// TwinCAT 3 PLC project SynergyPLC
// ProgramVersion: 3.1.4024.12
// libraries:
//   Tc2_EtherCAT, * (Beckhoff Automation GmbH)
//   Tc2_Standard, * (Beckhoff Automation GmbH)
//   Tc2_System, * (Beckhoff Automation GmbH)
//   Tc3_EventLogger, * (Beckhoff Automation GmbH)
//   Tc3_Module, * (Beckhoff Automation GmbH)
//   Tc3_PlasticInterfaceMotion, * (Beckhoff Automation GmbH)
//   Tc3_PlasticInterfaceNc, * (Beckhoff Automation GmbH)
// project tree:
//   GlobalBase/ WatchdogTimer.TcPOU
//   MotionControlBaseAnkur/ AxisBase.TcPOU (excluded from build), ModuleBase.TcPOU (not stored)
//   MotionControlBaseAnkur/DUTs/ Application.TcDUT, AxisData.TcDUT (excluded from build), AxisProperties.TcDUT, AxisStatus.TcDUT (not stored) (excluded from build), GearingType.TcDUT (not stored), Hardware.TcDUT (not stored), HomeFlagType.TcDUT, Homing.TcDUT, HomingMode.TcDUT (not stored), ID.TcDUT, ManualSettings.TcDUT, Mechanical.TcDUT (not stored), OperationLimits.TcDUT (excluded from build), OperationMode.TcDUT (excluded from build), StageBase.TcDUT, StepBase.TcDUT
//   MotionControlBaseAnkur/GVLs/ mcGlobal.TcGVL
//   MotionControlBase/DUTs/ ST_mcAxisNC.TcDUT, E_mcOperationMode.TcTLEO, ST_mcAxisStatus.TcDUT, ST_mcJogAllowance.TcDUT, ST_mcJogParameters.TcDUT, ST_mcAxisOperationLimits.TcDUT
//   MotionControlBase/ FB_mcModulesConfigurator.TcPOU, FB_mcAxisBase.TcPOU, FB_mcAxesConfigurator.TcPOU, FB_mcModuleBase.TcPOU, FB_mcOperationMode.TcPOU
//   MotionControlBase/GVLs/ mcGVL.TcGVL
//   Synergy/GVLs/ synGlobal.TcGVL
//   Synergy/MAIN/ Main1ms.TcPOU
//   / Task1ms.TcTTO
// real-time tasks:
//   TASK Task1ms: cycle T#1ms, priority 1, ADS port 351
// motion (NC):
//   TASK NC-Task 1 SAF: cycle T#1ms, priority 4, ADS port 501
//   TASK NC-Task 1 SVB: cycle T#1ms, priority 8, ADS port 511
//   AXIS Axis 1 (id 1)
//     OtherSettings: AllowMotionCmdToSlave=true
//     encoder EncType=1
//     drive DrvType=5
//       Analog: TorqueSetpointScale=10, ScaleFactorActTorque=0.1
//       TimeComp: TaskDelayCycles=1
//     controller CtrType=1
//       CtrPara: PriorControlFactor=1
//         Observer: BandWidth=20
//   AXIS Axis 2 (id 2)
//     OtherSettings: AllowMotionCmdToSlave=true
//     encoder EncType=1
//     drive DrvType=5
//       Analog: TorqueSetpointScale=10, ScaleFactorActTorque=0.1
//       TimeComp: TaskDelayCycles=1
//     controller CtrType=1
//       CtrPara: PriorControlFactor=1
//         Observer: BandWidth=20
//   AXIS Axis 3 (id 3)
//     OtherSettings: AllowMotionCmdToSlave=true
//     encoder EncType=1
//     drive DrvType=5
//       Analog: TorqueSetpointScale=10, ScaleFactorActTorque=0.1
//       TimeComp: TaskDelayCycles=1
//     controller CtrType=1
//       CtrPara: PriorControlFactor=1
//         Observer: BandWidth=20
//   AXIS Axis 4 (id 4)
//     OtherSettings: AllowMotionCmdToSlave=true
//     encoder EncType=1
//     drive DrvType=5
//       Analog: TorqueSetpointScale=10, ScaleFactorActTorque=0.1
//       TimeComp: TaskDelayCycles=1
//     controller CtrType=1
//       CtrPara: PriorControlFactor=1
//         Observer: BandWidth=20
//   AXIS Axis 5 (id 5)
//     OtherSettings: AllowMotionCmdToSlave=true
//     encoder EncType=1
//     drive DrvType=5
//       Analog: TorqueSetpointScale=10, ScaleFactorActTorque=0.1
//       TimeComp: TaskDelayCycles=1
//     controller CtrType=1
//       CtrPara: PriorControlFactor=1
//         Observer: BandWidth=20
//   AXIS Axis 6 (id 6)
//     OtherSettings: AllowMotionCmdToSlave=true
//     encoder EncType=1
//     drive DrvType=5
//       Analog: TorqueSetpointScale=10, ScaleFactorActTorque=0.1
//       TimeComp: TaskDelayCycles=1
//     controller CtrType=1
//       CtrPara: PriorControlFactor=1
//         Observer: BandWidth=20
//   AXIS Axis 7 (id 7)
//     OtherSettings: AllowMotionCmdToSlave=true
//     encoder EncType=1
//     drive DrvType=5
//       Analog: TorqueSetpointScale=10, ScaleFactorActTorque=0.1
//       TimeComp: TaskDelayCycles=1
//     controller CtrType=1
//       CtrPara: PriorControlFactor=1
//         Observer: BandWidth=20
//   AXIS Axis 8 (id 8)
//     OtherSettings: AllowMotionCmdToSlave=true
//     encoder EncType=1
//     drive DrvType=5
//       Analog: TorqueSetpointScale=10, ScaleFactorActTorque=0.1
//       TimeComp: TaskDelayCycles=1
//     controller CtrType=1
//       CtrPara: PriorControlFactor=1
//         Observer: BandWidth=20
// variable links:
//   SynergyPLC/SynergyPLC Instance <-> NC-Task 1 SAF/Axes/Axis 1
//     Task1ms Inputs/Main1ms.mcModules[1].Axis[1].fbLocalNc.AxisRef.NcToPlc <-> Outputs/ToPlc
//     Task1ms Outputs/Main1ms.mcModules[1].Axis[1].fbLocalNc.AxisRef.PlcToNc <-> Inputs/FromPlc
//   SynergyPLC/SynergyPLC Instance <-> NC-Task 1 SAF/Axes/Axis 2
//     Task1ms Inputs/Main1ms.mcModules[1].Axis[2].fbLocalNc.AxisRef.NcToPlc <-> Outputs/ToPlc
//     Task1ms Outputs/Main1ms.mcModules[1].Axis[2].fbLocalNc.AxisRef.PlcToNc <-> Inputs/FromPlc
//   SynergyPLC/SynergyPLC Instance <-> NC-Task 1 SAF/Axes/Axis 3
//     Task1ms Inputs/Main1ms.mcModules[1].Axis[3].fbLocalNc.AxisRef.NcToPlc <-> Outputs/ToPlc
//     Task1ms Outputs/Main1ms.mcModules[1].Axis[3].fbLocalNc.AxisRef.PlcToNc <-> Inputs/FromPlc
//   SynergyPLC/SynergyPLC Instance <-> NC-Task 1 SAF/Axes/Axis 4
//     Task1ms Inputs/Main1ms.mcModules[1].Axis[4].fbLocalNc.AxisRef.NcToPlc <-> Outputs/ToPlc
//     Task1ms Outputs/Main1ms.mcModules[1].Axis[4].fbLocalNc.AxisRef.PlcToNc <-> Inputs/FromPlc
//   SynergyPLC/SynergyPLC Instance <-> NC-Task 1 SAF/Axes/Axis 5
//     Task1ms Inputs/Main1ms.mcModules[1].Axis[5].fbLocalNc.AxisRef.NcToPlc <-> Outputs/ToPlc
//     Task1ms Outputs/Main1ms.mcModules[1].Axis[5].fbLocalNc.AxisRef.PlcToNc <-> Inputs/FromPlc
//   SynergyPLC/SynergyPLC Instance <-> NC-Task 1 SAF/Axes/Axis 6
//     Task1ms Inputs/Main1ms.mcModules[1].Axis[6].fbLocalNc.AxisRef.NcToPlc <-> Outputs/ToPlc
//     Task1ms Outputs/Main1ms.mcModules[1].Axis[6].fbLocalNc.AxisRef.PlcToNc <-> Inputs/FromPlc
//   SynergyPLC/SynergyPLC Instance <-> NC-Task 1 SAF/Axes/Axis 7
//     Task1ms Inputs/Main1ms.mcModules[1].Axis[7].fbLocalNc.AxisRef.NcToPlc <-> Outputs/ToPlc
//     Task1ms Outputs/Main1ms.mcModules[1].Axis[7].fbLocalNc.AxisRef.PlcToNc <-> Inputs/FromPlc
//   SynergyPLC/SynergyPLC Instance <-> NC-Task 1 SAF/Axes/Axis 8
//     Task1ms Inputs/Main1ms.mcModules[1].Axis[8].fbLocalNc.AxisRef.NcToPlc <-> Outputs/ToPlc
//     Task1ms Outputs/Main1ms.mcModules[1].Axis[8].fbLocalNc.AxisRef.PlcToNc <-> Inputs/FromPlc

CONFIGURATION SynergyPLC
    RESOURCE PLC ON TwinCAT3
        TASK Task1ms(INTERVAL := T#1ms, PRIORITY := 1);
        PROGRAM Main1ms WITH Task1ms : Main1ms;
    END_RESOURCE
END_CONFIGURATION

// ---- MotionControlBaseAnkur/DUTs/Application.TcDUT
TYPE Application :
STRUCT
	GearingType			:	GearingType;
END_STRUCT
END_TYPE

// ---- MotionControlBaseAnkur/DUTs/AxisData.TcDUT
TYPE AxisData :
STRUCT
	lrActPosition			:		LREAL;
	lrActVelocity			:		LREAL;
	lrActTorque				:		LREAL;
	lrMotorTemp				:		LREAL;
END_STRUCT
END_TYPE

// ---- MotionControlBaseAnkur/DUTs/AxisProperties.TcDUT
TYPE AxisProperties :
STRUCT
	stIdentification			:		ID;
	stHardware					:		Hardware;
	stApplication				:		Application;
	stHoming					:		Homing;
	stOperationLimits			:		OperationLimits;
END_STRUCT
END_TYPE

// ---- MotionControlBaseAnkur/DUTs/HomeFlagType.TcDUT
{attribute 'qualified_only'}
{attribute 'strict'}
TYPE HomeFlagType :
(
	eSensor := 1,
	eHardStop := 2
);
END_TYPE

// ---- MotionControlBaseAnkur/DUTs/Homing.TcDUT
TYPE Homing :
STRUCT
	Mode			:		HomingMode;
	FlagType		:		HomeFlagType;
	bHomeInput		:		BOOL;
	rOffset			:		REAL;
	rVelocity		:		REAL;
	rTorque			:		REAL;
END_STRUCT
END_TYPE

// ---- MotionControlBaseAnkur/DUTs/ID.TcDUT
TYPE ID :
STRUCT
	intIndex			:	INT;
	sName				:	STRING;
	intMasterIndex		:	INT;
END_STRUCT
END_TYPE

// ---- MotionControlBaseAnkur/DUTs/ManualSettings.TcDUT
TYPE ManualSettings :
STRUCT
	lrJogVelocity			:		LREAL;
	lrJogRamp				:		LREAL;
	lrJogJerk				:		LREAL;
	lrJogTorque				:		LREAL;
END_STRUCT
END_TYPE

// ---- MotionControlBaseAnkur/DUTs/OperationLimits.TcDUT
TYPE OperationLimits :
STRUCT
	rMinPosition		:		REAL;
	rMaxPosition		:		REAL;
	rMaxVelocity		:		REAL;
	rJogVelocity		:		REAL;
	tMaxMotionTime		:		TIME;
END_STRUCT
END_TYPE

// ---- MotionControlBaseAnkur/DUTs/OperationMode.TcDUT
{attribute 'qualified_only'}
{attribute 'strict'}
TYPE OperationMode :
(
	eManual 	:= 1,
	eService 	:= 2,
	eAutomatic 	:= 3,
	eSimulation := 4
);
END_TYPE

// ---- MotionControlBaseAnkur/DUTs/StageBase.TcDUT
TYPE StageBase :
STRUCT
	bEnable			:		BOOL;
	bTrigger		:		BOOL;
	bMoveActive		:		BOOL;
	tMoveTime		:		TIME;
	intSteps		:		INT;
	Step			:		ARRAY[1..5] OF StepBase;
END_STRUCT
END_TYPE

// ---- MotionControlBaseAnkur/DUTs/StepBase.TcDUT
TYPE StepBase :
STRUCT
	rSetVelocity		:		REAL;
	rSetRamp			:		REAL;
	rSetEndPosition		:		REAL;
END_STRUCT
END_TYPE

// ---- MotionControlBase/DUTs/ST_mcAxisNC.TcDUT
TYPE ST_mcAxisNC :
STRUCT
	lrActPosition			:		LREAL;
	lrActVelocity			:		LREAL;
	lrActTorque				:		LREAL;
	lrMotorTemp				:		LREAL;
END_STRUCT
END_TYPE

// ---- MotionControlBase/DUTs/E_mcOperationMode.TcTLEO
{attribute 'qualified_only'}
{attribute 'strict'}
TYPE E_mcOperationMode : // Operation modes defined
(
	Initialization :=1,
	Service :=2,
	Manual :=3,
	Simulation :=4,
	Automatic :=5
);
END_TYPE

// ---- MotionControlBase/DUTs/ST_mcAxisStatus.TcDUT
TYPE ST_mcAxisStatus :
STRUCT
	bPowerEnabled		:		BOOL; // Power is enabled
	bHomed				:		BOOL; // Homed
	bStandStill			:		BOOL; // Standstill
	bMoving				: 		BOOL; // Moving
	bError				:       BOOL; // Error
END_STRUCT
END_TYPE

// ---- MotionControlBase/DUTs/ST_mcJogAllowance.TcDUT
TYPE ST_mcJogAllowance :
STRUCT
	bAllowJogParameters : BOOL; // Boolean to check if jogging is allowed because of parameters
	bAllowJogOperationMode : BOOL; // Boolean to check if jogging is allowed because of operation mode
END_STRUCT
END_TYPE

// ---- MotionControlBase/DUTs/ST_mcJogParameters.TcDUT
TYPE ST_mcJogParameters :
STRUCT
	lrJogAcceleration		:			LREAL;	//Jog acceleration
	lrJogDeceleration		: 			LREAL;	//Jog deceleration
	lrJogJerkValue			:			LREAL;	//Jog jerk
	lrJogVelocity			:			LREAL;	//Jog velocity
	lrJogLimitPositive		:      		LREAL;  // Jog Positive Torque Limit
	lrJogLimitNegative		:			LREAL;  // Jog Negative Torque Limit
END_STRUCT
END_TYPE

// ---- MotionControlBase/DUTs/ST_mcAxisOperationLimits.TcDUT
TYPE ST_mcAxisOperationLimits :
STRUCT
	lrSoftMinPosition	:			LREAL;	//Minimum position of travel allowed
	lrSoftMaxPosition	: 			LREAL;	//Maximum position of travel allowed
	lrDefaultAcceleration	:		LREAL;	//Maximum Acceleration allowed
	lrDefaultDeceleration	:		LREAL;	//Minimum deceleration allowed
	lrMaxVelocity		:      		LREAL;  //Maximum Velocity allowed
END_STRUCT
END_TYPE

// ---- MotionControlBaseAnkur/GVLs/mcGlobal.TcGVL
{attribute 'qualified_only'}
VAR_GLOBAL
//	fbMotionModule	:		ARRAY[1..cMaxNoOfModule] OF ModuleBase;
END_VAR

VAR_GLOBAL CONSTANT
	cMaxNoOfAxis			:		INT := 8;
	cMinNoOfAxis			:		INT := 1;
	
	cMaxNoOfModule			:		INT := 4;
	cMinNoOfModule			:		INT := 1;
	
	
END_VAR

// ---- MotionControlBase/GVLs/mcGVL.TcGVL
{attribute 'qualified_only'}
VAR_GLOBAL
	OperationMode : FB_MCOperationMode; // Operation mode 
	AxesConfigurator : FB_mcAxesConfigurator; // Configurator to set number of axes
	ModulesConfigurator : FB_mcModulesConfigurator; // Configurator to set number of modules
END_VAR

VAR_GLOBAL CONSTANT
	cMaxAxesCapacity: UINT := 8; // Maximum designed axes capacity by hardware
	cMinAxesCapacity: UINT := 1; // Minimum designed axes capacity by hardware
	cMaxModuleCapacity	: UINT := 4; // Maximum designed modules capacity by hardware
	cMinModuleCapacity	: UINT := 1; // Minimum designed modules capacity by hardware
END_VAR

// ---- Synergy/GVLs/synGlobal.TcGVL
{attribute 'qualified_only'}
VAR_GLOBAL
END_VAR

// ---- Synergy/MAIN/Main1ms.TcPOU
PROGRAM Main1ms
VAR
	mcModules		: ARRAY [1..mcGvl.cMaxModuleCapacity] OF FB_mcModuleBase;
	mcCount			: UINT;
END_VAR

A_mcCyclic();

ACTION A_mcCyclic:
mcGvl.OperationMode(); // Operation mode 
mcGvl.AxesConfigurator(); // Configurator to set number of axes
mcGvl.ModulesConfigurator(); // Configurator to set number of modules

FOR mcCount := 1 TO mcGvl.ModulesConfigurator.uiNoModulesActive DO
	mcModules[mcCount]();
END_FOR;
END_ACTION

END_PROGRAM

// ---- MotionControlBase/FB_mcModuleBase.TcPOU
FUNCTION_BLOCK FB_mcModuleBase
VAR
	Axis			:		ARRAY[1..mcGvl.cMaxAxesCapacity] OF FB_mcAxisBase[
															(AxisName		:=	'Axis1',
															nPtpPoints		:=	5,
															iProcessHandler	:=	0,
															iTorqueLimiting	:=	0,
															iPosCamLookup	:=	0,
															iVeloCamLookup	:=	0,
															iPtpCamLookup	:=	0),
															(AxisName		:=	'Axis2',
															nPtpPoints		:=	5,
															iProcessHandler	:=	0,
															iTorqueLimiting	:=	0,
															iPosCamLookup	:=	0,
															iVeloCamLookup	:=	0,
															iPtpCamLookup	:=	0),
															(AxisName		:=	'Axis3',
															nPtpPoints		:=	5,
															iProcessHandler	:=	0,
															iTorqueLimiting	:=	0,
															iPosCamLookup	:=	0,
															iVeloCamLookup	:=	0,
															iPtpCamLookup	:=	0),
															(AxisName		:=	'Axis4',
															nPtpPoints		:=	5,
															iProcessHandler	:=	0,
															iTorqueLimiting	:=	0,
															iPosCamLookup	:=	0,
															iVeloCamLookup	:=	0,
															iPtpCamLookup	:=	0),
															(AxisName		:=	'Axis5',
															nPtpPoints		:=	5,
															iProcessHandler	:=	0,
															iTorqueLimiting	:=	0,
															iPosCamLookup	:=	0,
															iVeloCamLookup	:=	0,
															iPtpCamLookup	:=	0),
															(AxisName		:=	'Axis6',
															nPtpPoints		:=	5,
															iProcessHandler	:=	0,
															iTorqueLimiting	:=	0,
															iPosCamLookup	:=	0,
															iVeloCamLookup	:=	0,
															iPtpCamLookup	:=	0),
															(AxisName		:=	'Axis7',
															nPtpPoints		:=	5,
															iProcessHandler	:=	0,
															iTorqueLimiting	:=	0,
															iPosCamLookup	:=	0,
															iVeloCamLookup	:=	0,
															iPtpCamLookup	:=	0),
															(AxisName		:=	'Axis8',
															nPtpPoints		:=	5,
															iProcessHandler	:=	0,
															iTorqueLimiting	:=	0,
															iPosCamLookup	:=	0,
															iVeloCamLookup	:=	0,
															iPtpCamLookup	:=	0)
															];
	uiCount				:		UINT;
END_VAR

VAR_INPUT
END_VAR

FOR uiCount := 1 TO mcGVL.AxesConfigurator.uiNoAxesActive DO
	Axis[uiCount].A_Cyclic();
END_FOR

END_FUNCTION_BLOCK

// ---- MotionControlBase/FB_mcAxisBase.TcPOU
FUNCTION_BLOCK FB_mcAxisBase EXTENDS FB_AxisNcBase
VAR_INPUT
	bPowerEnable : BOOL; // Enable Power
	bJogPositive : BOOL; // Jog Positive
	bJogNegative : BOOL; // Jog Negative
	bStop: BOOL; // Stop axis
	bReset: BOOL; // Reset axis
	bExecuteOpLimits: BOOL; // Write operation limits
END_VAR
VAR_OUTPUT
	bBaseFBError : BOOL; // Internal library error
	stStatus: ST_mcAxisStatus; // Status booleans of Axis
	stDataNC: ST_mcAxisNC; // Real data from drive
END_VAR
VAR
	stJogAllowance : ST_mcJogAllowance; // Status bits troubleshooting
	rTrigOpLimits : R_TRIG; // Operation limits trigger
END_VAR

VAR_INPUT PERSISTENT
	stJogParameters : ST_mcJogParameters; // Accel, Decel, Velocity etc
	stOperationLimits : ST_mcAxisOperationLimits; // Soft pos limits, vel limits
END_VAR

VAR CONSTANT 
	cJogMinParameter : REAL := 0.0;  // Minimum parameters for jog to be set to 0 
END_VAR

A_Cyclic(); // Cyclic calls of routines

ACTION A_Cyclic:
SUPER^.Cyclic();						//Cyclic method to initialize underlying motion blocks

IF M_FbError() THEN
;  // Error Exists in Base FB
ELSE  

	// Calling of method to turn power on/off
	M_Power(bCommand:= bPowerEnable);  		
	
	//Calling of method to jog + or - 
	M_Jog(bCommandJogP:= bJogPositive,bCommandJogM:= bJogNegative);

END_IF;

// Calling of method to stop axis
M_Stop(bCommand:= bStop); 

// Calling of method to reset axis
M_Reset(bCommand:= bReset); 

// Calling of method to write operation limits of an axis
rTrigOpLimits(CLK:= bExecuteOpLimits);
M_OperationLimits(bCommand:= rTrigOpLimits.Q);

// Axis Status bits
A_Status();

//Axis Real Data
A_DataNC();
END_ACTION

ACTION A_DataNC:
(*
Data from drive
*)

THIS^.stDataNC.lrActPosition:= SUPER^.ActualsNc.Position;
THIS^.stDataNC.lrActVelocity:= SUPER^.ActualsNc.Velocity;
THIS^.stDataNC.lrActTorque:= SUPER^.ActualsNc.Torque;
//TODO: THIS^.stDataNC.lrMotorTemp:= ;
END_ACTION

ACTION A_Status:
(*
Status bits for axis
*)

THIS^.stStatus.bPowerEnabled:= THIS^.Power.Status;
THIS^.stStatus.bStandStill:= SUPER^.fbLocalNc.AxisRef.Status.StandStill;
THIS^.stStatus.bMoving:= SUPER^.fbLocalNc.AxisRef.Status.Moving;
THIS^.stStatus.bHomed:= SUPER^.fbLocalNc.AxisRef.Status.Homed;
THIS^.stStatus.bError:= SUPER^.fbLocalNc.AxisRef.Status.Error;
END_ACTION

METHOD M_FbError : BOOL
VAR_INPUT
END_VAR
IF bError THEN
	bBaseFBError := TRUE;			//Set bErrorChk to TRUE so none of the other methods are called
	M_FbError :=TRUE;
ELSE
	bBaseFBError := FALSE;
	M_FbError :=FALSE;
END_IF
END_METHOD

METHOD M_Jog : HRESULT
VAR_INPUT
	bCommandJogP 	:   BOOL;
	bCommandJogM	:	BOOL;
END_VAR

VAR 
	
END_VAR
// ======================================================================
IF bCommandJogP OR bCommandJogM THEN

	IF M_JogPreChecks() THEN // Calls to check pre conditions to allow jogging
		F_SucceededHr(Jog.SetParameter(fAcceleration:=stJogParameters.lrJogAcceleration, fDeceleration:=stJogParameters.lrJogDeceleration,
		fJerk:=stJogParameters.lrJogJerkValue,fVelocity:=stJogParameters.lrJogVelocity), M_Jog);

					IF bCommandJogP THEN
					 F_SucceededHr(Jog.DoJogP(bExecute:=TRUE),M_Jog);	
					ELSIF bCommandJogM THEN
			 		 F_SucceededHr(Jog.DoJogM(bExecute:=TRUE),M_Jog);
					ELSE
					F_SucceededHr(Jog.DoJogP(bExecute:=FALSE),M_Jog); // Stop the jog when + or - button is released
					F_SucceededHr(Jog.DoJogM(bExecute:=FALSE),M_Jog); 
					END_IF
	ELSE
		F_SucceededHr(Jog.DoJogP(bExecute:=FALSE),M_Jog); // Stop the jog if pre conditions are not met even during motion 
		F_SucceededHr(Jog.DoJogM(bExecute:=FALSE),M_Jog);
	END_IF
ELSE
			F_SucceededHr(Jog.DoJogP(bExecute:=FALSE),M_Jog); // Stop the jog when its not + or - button  
			F_SucceededHr(Jog.DoJogM(bExecute:=FALSE),M_Jog);
END_IF		
	
// ======================================================================
END_METHOD

METHOD M_JogPreChecks : BOOL
VAR_INPUT
END_VAR
VAR
END_VAR
IF MCgvl.OperationMode.eModeActive = E_mcOperationMode.Manual THEN
	stJogAllowance.bAllowJogOperationMode:=TRUE;
//	fbMsgJogOperationMode.Release();
	ELSE
//	fbMsgJogOperationMode.SendMessage(TC_Events.TC_EventJog.OperationMode,'Change Operation Mode');
    stJogAllowance.bAllowJogOperationMode:=FALSE;	
END_IF

IF stJogParameters.lrJogAcceleration > cJogMinParameter AND stJogParameters.lrJogDeceleration > cJogMinParameter AND stJogParameters.lrJogVelocity > cJogMinParameter THEN 
	stJogAllowance.bAllowJogParameters:=TRUE;
//	fbMsgJogParamters.Release();
	ELSE
//	fbMsgJogParamters.SendMessage(TC_Events.TC_EventJog.Parameters,'Check Acceleration, Decceleration and Velocity');
    stJogAllowance.bAllowJogParameters:=FALSE;	
END_IF

M_JogPreChecks:= stJogAllowance.bAllowJogOperationMode AND stJogAllowance.bAllowJogParameters;
END_METHOD

METHOD M_OperationLimits : BOOL
VAR_INPUT
	bCommand		:		BOOL;
END_VAR
IF bCommand THEN
	THIS^.MotionParams.SoftEndMax :=stOperationLimits.lrSoftMaxPosition;
	THIS^.MotionParams.SoftEndMin :=stOperationLimits.lrSoftMinPosition;
	THIS^.MotionParams.MaxAcceleration:=stOperationLimits.lrDefaultAcceleration;
	THIS^.MotionParams.MaxDeceleration:=stOperationLimits.lrDefaultDeceleration;
	THIS^.MotionParams.MaxVeloApplication:=stOperationLimits.lrMaxVelocity;
	bExecuteOpLimits:= FALSE; 
END_IF
END_METHOD

METHOD M_Power : HRESULT
VAR_INPUT
	bCommand : BOOL;
END_VAR

VAR
END_VAR
// ======================================================================

	IF bCommand THEN
		IF F_SucceededHr(Power.FeedEnable(bFeedEnaPositive:=TRUE,bFeedEnaNegative:=TRUE), M_Power) THEN
			F_SucceededHr(Power.DoPower(bEnable:=TRUE), M_Power);
		END_IF

	
	ELSIF NOT bCommand THEN
		IF F_SucceededHr(Power.FeedEnable(bFeedEnaPositive:=FALSE,bFeedEnaNegative:=FALSE), M_Power) THEN
			F_SucceededHr(Power.DoPower(bEnable:=FALSE), M_Power);
		END_IF
	
	ELSE 
		; // cyclic calls of this method 
	END_IF		
// ======================================================================
END_METHOD

METHOD M_Reset : HRESULT
VAR_INPUT
	bCommand : BOOL;
END_VAR

VAR
END_VAR
// ======================================================================

	IF bCommand THEN
		IF F_SucceededHr(Reset.DoReset(bExecute:=TRUE), M_Reset) THEN
			bError:=FALSE;
		END_IF
	
	ELSIF NOT bCommand THEN		
		F_SucceededHr(Reset.DoReset(bExecute:=FALSE), M_Reset);
		
	ELSE 
		; // cyclic calls of this method 
	END_IF
		
// ======================================================================
END_METHOD

METHOD M_Stop : HRESULT
VAR_INPUT
	bCommand : BOOL;
END_VAR

VAR
END_VAR
// ======================================================================

	IF bCommand THEN
//		bMovePtpAxis := FALSE;
		F_SucceededHr(Stop.DoStop(bExecute:=TRUE), M_Stop);
	
	ELSIF NOT bCommand THEN
		F_SucceededHr(Stop.DoStop(bExecute:=FALSE), M_Stop);
		
	ELSE 
		; // cyclic calls of this method 
	END_IF
		
// ======================================================================
END_METHOD

END_FUNCTION_BLOCK

// ---- MotionControlBase/FB_mcOperationMode.TcPOU
FUNCTION_BLOCK FB_mcOperationMode
VAR_INPUT
	eModeRequired : E_mcOperationMode;
END_VAR
VAR_OUTPUT
	eModeActive  : E_mcOperationMode;
END_VAR
VAR
	//	fbMsgAutomaticMode : FB_Messagess;
END_VAR

M_SetMode(eCommand := eModeRequired);

METHOD M_PreCheckAutomatic : BOOL
VAR_INPUT
END_VAR
(*IF Main.fbAxis.Power.Status THEN
	M_PreCheckAutomatic:=TRUE;
//	fbMsgAutomaticMode.Release();
	ELSE
//	fbMsgAutomaticMode.SendMessage(TC_Events.TC_EventOperationModeAutomatic.AxisPower,'');
    M_PreCheckAutomatic:=FALSE;	
END_IF
*);
END_METHOD

METHOD M_SetMode : HRESULT
VAR_INPUT
	eCommand : E_mcOperationMode;
END_VAR
CASE eCommand OF 
	
E_mcOperationMode.Initialization :
	THIS^.eModeActive:=E_mcOperationMode.Initialization;
	M_SetMode:=F_HRESULTSUCCESS(NOERR);

E_mcOperationMode.Service :
	THIS^.eModeActive:=E_mcOperationMode.Service;
	M_SetMode:=F_HRESULTSUCCESS(NOERR);

E_mcOperationMode.Manual:
	THIS^.eModeActive:=E_mcOperationMode.Manual;
	M_SetMode:=F_HRESULTSUCCESS(NOERR);

E_mcOperationMode.Simulation:
	THIS^.eModeActive:=E_mcOperationMode.Simulation;
	M_SetMode:=F_HRESULTSUCCESS(NOERR);

E_mcOperationMode.Automatic:
	IF M_PreCheckAutomatic () THEN
		THIS^.eModeActive:=E_mcOperationMode.Automatic;
		M_SetMode:=F_HRESULTSUCCESS(NOERR);
	ELSE
		THIS^.eModeRequired:=THIS^.eModeActive;
		M_SetMode:=F_HRESULTFAILURE(DEVICE_NOTREADY);
	END_IF	

ELSE
	M_SetMode:=F_HRESULTFAILURE(DEVICE_INVALIDDATA);

END_CASE
END_METHOD

END_FUNCTION_BLOCK

// ---- MotionControlBase/FB_mcAxesConfigurator.TcPOU
FUNCTION_BLOCK FB_mcAxesConfigurator
VAR_INPUT
	bExecute : BOOL; // Boolean to execute the function block
	uiNoAxesRequired : UINT:= 1; // Get from user no of axes he wants to use
	sNetId: T_AmsNetId;
	pArrEcScannedSlaveInfo: POINTER TO ARRAY [0..EC_MAX_SLAVES] OF ST_EcSlaveScannedData;
	cbBufLen: UDINT;
	tTimeout: TIME;
END_VAR
VAR_OUTPUT
	uiNoAxesActive : UINT; // current no of active axes
	bNoOfAxesMatched : BOOL; // Entered no of axes matched with ECAT ring axes available
END_VAR

VAR
	uiECATScannedAxes: UINT; // Scan the ECAT ring to find the no of axis available
	fbScannedAxes	: FB_ECGETSCANNEDSLAVES;
	rTrigExecute	: R_TRIG;
END_VAR

(*Axis configurator is designed to get number of axis from user and scan ECAT 
TODO: Add further elements to it
*)

rTrigExecute(CLK:= bExecute);
M_NoOfAxes(bCommand:= rTrigExecute.Q);

METHOD M_NoOfAxes : BOOL
VAR_INPUT
	bCommand : BOOL; 
END_VAR
IF bCommand THEN

	fbScannedAxes(
		bExecute:= TRUE, 
		sNetId:= sNetId, 
		pArrEcScannedSlaveInfo:= pArrEcScannedSlaveInfo, 
		cbBufLen:= cbBufLen, 
		tTimeout:= tTimeout ,  
		nSlaves=> uiECATScannedAxes);

	IF (uiNoAxesRequired <> uiNoAxesActive) OR (uiNoAxesRequired <> uiECATScannedAxes) THEN
		
		IF (uiNoAxesRequired < mcGvl.cMinAxesCapacity) OR (uiNoAxesRequired > mcGvl.cMaxAxesCapacity) THEN
			; //TODO: Entered no of axes are not possible set the message to user
	//	ELSIF (uiNoAxesRequired <> uiECATScannedAxes) THEN
	//		bNoOfAxesMatched:=FALSE; // Entered no of axes are not matching the ECAT ring axes available
		ELSE
			uiNoAxesActive:= uiNoAxesRequired; // Set the required number of axes to active no of axes
			bNoOfAxesMatched:= TRUE;	
		END_IF
	
	ELSE
		; // cyclic calls for inequality
	END_IF
	// Reset the input of Function block so next time it has to look for only rising edge
	bExecute:= FALSE; 
ELSE
	fbScannedAxes(bExecute:= FALSE); // cyclic calls for bCommand
END_IF

M_NoOfAxes:= bNoOfAxesMatched;
END_METHOD

END_FUNCTION_BLOCK

// ---- MotionControlBase/FB_mcModulesConfigurator.TcPOU
FUNCTION_BLOCK FB_mcModulesConfigurator
VAR_INPUT
	bExecute : BOOL; // Execute the function block
	uiNoModulesRequired : UINT:= 1; // Enter modules required
	sNetId: T_AmsNetId;
	pArrEcScannedSlaveInfo: POINTER TO ARRAY [0..EC_MAX_SLAVES] OF ST_EcSlaveScannedData;
	cbBufLen: UDINT;
	tTimeout: TIME;
END_VAR
VAR_OUTPUT
	uiNoModulesActive : UINT; // current no of active axes
	bNoOfModulesMatched : BOOL; // Entered no of axes matched with ECAT ring axes available
END_VAR

VAR
	uiECATScannedModules: UINT; // Scan the ECAT ring to find the no of axis available
	fbScannedModules	: FB_ECGETSCANNEDSLAVES;
	rTrigExecute		: R_TRIG;
END_VAR

(*Axis configurator is designed to get number of axis from user and scan ECAT 
TODO: Add further elements to it
*)

rTrigExecute(CLK:= bExecute);
M_NoOfModules(bCommand:= rTrigExecute.Q);

METHOD M_NoOfModules : BOOL
VAR_INPUT
	bCommand : BOOL; 
END_VAR
IF bCommand THEN

	fbScannedModules(
		bExecute:= TRUE, 
		sNetId:= sNetId, 
		pArrEcScannedSlaveInfo:= pArrEcScannedSlaveInfo, 
		cbBufLen:= cbBufLen, 
		tTimeout:= tTimeout ,  
		nSlaves=> uiECATScannedModules);

	IF (uiNoModulesRequired <> uiNoModulesActive) OR (uiNoModulesRequired <> uiECATScannedModules) THEN
		
		IF (uiNoModulesRequired < mcGvl.cMinModuleCapacity) OR (uiNoModulesRequired > mcGvl.cMaxModuleCapacity) THEN
			; //TODO: Entered no of axes are not possible set the message to user
	//	ELSIF (uiNoModulesRequired <> uiECATScannedModules) THEN
	//		bNoOfModulesMatched:=FALSE; // Entered no of axes are not matching the ECAT ring axes available
		ELSE
			uiNoModulesActive:= uiNoModulesRequired; // Set the required number of axes to active no of axes
			bNoOfModulesMatched:= TRUE;	
		END_IF
	
	ELSE
		; // cyclic calls for inequality
	END_IF
	// Reset the input of Function block so next time it has to look for only rising edge
	bExecute:= FALSE; 
ELSE
	fbScannedModules(bExecute:= FALSE); // cyclic calls for bCommand
END_IF

M_NoOfModules:= bNoOfModulesMatched;
END_METHOD

END_FUNCTION_BLOCK

// ---- GlobalBase/WatchdogTimer.TcPOU
FUNCTION_BLOCK WatchdogTimer
VAR_INPUT
END_VAR
VAR_OUTPUT
END_VAR
VAR
END_VAR

END_FUNCTION_BLOCK

// ---- MotionControlBaseAnkur/AxisBase.TcPOU
FUNCTION_BLOCK AxisBase EXTENDS FB_AxisNcBase
VAR_INPUT
	bEnablePower		:		BOOL;
	bJogPositive		:		BOOL;
	bJogNegative		:		BOOL;
	Command				:		BYTE;
	stManualSettings	:		ManualSettings;
END_VAR

VAR_OUTPUT
	stData				:		AxisData;
	stStatus			:		AxisStatus;
	Status				:		BYTE;
END_VAR

VAR
	stProperties		:		AxisProperties;
	stPtpStage			:		ARRAY[1..4] OF StageBase;
	tWatchdogTimer		:		TIME;
	fbWatchdogTimer		:		WatchdogTimer;
END_VAR

ACTION A_Cyclic:
//Cyclic method to initialize underlying motion blocks
SUPER^.Cyclic();

A_MeasureData();

M_ServoPower(bEnablePower := bEnablePower);

M_MoveJog(bJogPositive := bJogPositive,
		bJogNegative := bJogNegative);
END_ACTION

ACTION A_Dummy:

END_ACTION

ACTION A_MeasureData:
THIS^.stData.lrActPosition := THIS^.ActualsNc.Position;
THIS^.stData.lrActVelocity := THIS^.ActualsNc.Velocity;
THIS^.stData.lrActTorque := THIS^.ActualsNc.Torque;

(*TO DO
THIS^.Data.lrMotorTemp :=
*)
END_ACTION

METHOD M_AutoTune : BOOL
VAR_INPUT
END_VAR
END_METHOD

METHOD M_CreepJog : BOOL
VAR_INPUT
END_VAR
END_METHOD

METHOD M_Home : BOOL
VAR_INPUT
END_VAR
END_METHOD

METHOD M_Init
VAR_INPUT
END_VAR
END_METHOD

METHOD M_JogToStartPos : BOOL
VAR_INPUT
END_VAR
END_METHOD

METHOD M_MarkHome : BOOL
VAR_INPUT
END_VAR
END_METHOD

METHOD M_MonitorLimits : BOOL
VAR_INPUT
END_VAR
END_METHOD

METHOD M_MoveJog : HRESULT
VAR_INPUT
	bJogPositive		:		BOOL;
	bJogNegative		:		BOOL;
END_VAR

VAR_OUTPUT
	bActive				:		BOOL;
END_VAR
IF bJogPositive OR bJogNegative THEN
	//Set Jog Parameters
	F_SucceededHr(Jog.SetParameter(fAcceleration := THIS^.stManualSettings.lrJogRamp,
								   fDeceleration := THIS^.stManualSettings.lrJogRamp,
								   fJerk := THIS^.stManualSettings.lrJogJerk,
								   fVelocity := THIS^.stManualSettings.lrJogVelocity), M_MoveJog);
	Jog.TorqueLimiting := stManualSettings.lrJogTorque;
	
	IF M_MoveJog_PreCheck() THEN
		//Execute Jog
		IF bJogPositive THEN
			F_SucceededHr(Jog.DoJogP(bExecute := TRUE), M_MoveJog);	
		ELSIF bJogNegative THEN
			F_SucceededHr(Jog.DoJogM(bExecute := TRUE), M_MoveJog);
		ELSE
			// Stop the jog when + or - button is released
			F_SucceededHr(Jog.DoJogP(bExecute := FALSE), M_MoveJog); 
			F_SucceededHr(Jog.DoJogM(bExecute := FALSE), M_MoveJog);
		END_IF
	ELSE
		F_SucceededHr(Jog.DoJogP(bExecute := FALSE), M_MoveJog);
		F_SucceededHr(Jog.DoJogM(bExecute := FALSE), M_MoveJog);
	END_IF
END_IF
END_METHOD

METHOD M_MoveJog_PreCheck : BOOL
VAR_INPUT
END_VAR

VAR
	bAllowJogOperationMode: BOOL;
END_VAR
(*
IF MCgvl.fbOperationMode.eModeActive = E_OperationMode.Manual THEN
	bAllowJogOperationMode:=TRUE;
//	fbMsgJogOperationMode.Release();
	ELSE
//	fbMsgJogOperationMode.SendMessage(TC_Events.TC_EventJog.OperationMode,'Change Operation Mode');
    bAllowJogOperationMode:=FALSE;	
END_IF

IF stJogParameters.lrJogAcceleration > crJogMinParameter AND stJogParameters.lrJogDeceleration > crJogMinParameter
AND stJogParameters.lrJogVelocity > crJogMinParameter THEN 
	bAllowJogParameters:=TRUE;
//	fbMsgJogParamters.Release();
	ELSE
//	fbMsgJogParamters.SendMessage(TC_Events.TC_EventJog.Parameters,'Check Acceleration, Decceleration and Velocity');
    bAllowJogParameters:=FALSE;	
END_IF

M_PreChecks:= bAllowJogOperationMode AND bAllowJogParameters;
*)
M_MoveJog_PreCheck := TRUE;
END_METHOD

METHOD M_MovePtp
VAR_INPUT
END_VAR
END_METHOD

METHOD M_ServoPower : HRESULT
VAR_INPUT
	bEnablePower	:		BOOL;
END_VAR

VAR_OUTPUT
	bDone			:		BOOL;
	bError			:		BOOL;					
END_VAR
IF bEnablePower THEN
	IF F_SucceededHr(Power.FeedEnable(bFeedEnaPositive:=TRUE,bFeedEnaNegative:=TRUE), M_ServoPower) THEN
	F_SucceededHr(Power.DoPower(bEnable:=TRUE), M_ServoPower);
	END_IF

ELSIF NOT bEnablePower THEN
	IF F_SucceededHr(Power.FeedEnable(bFeedEnaPositive:=FALSE,bFeedEnaNegative:=FALSE), M_ServoPower) THEN
	F_SucceededHr(Power.DoPower(bEnable:=FALSE), M_ServoPower);
	END_IF

ELSE 
	; // cyclic calls of this method 
END_IF
END_METHOD

METHOD M_StopMotion : HRESULT
VAR_INPUT
END_VAR
F_SucceededHr(Stop.DoStop(bExecute := TRUE), M_StopMotion);
END_METHOD

METHOD M_StrokeCheck : BOOL
VAR_INPUT
END_VAR
END_METHOD

END_FUNCTION_BLOCK
